(* Logix 5000 project; controller APM vendor 1 type 14 code 156 rev 30.11; software revision 30.00 *)

TASK MainTask (continuous, watchdog 500 ms) : MainProgram

MODULES
   Local : vendor 1 type 14 code 156 (Compact 0, rev 30.11)
END_MODULES

PROGRAM MainProgram   (* main routine MainRoutine *)
VAR
   CT_ACT_CT0 : BOOL;
   CT_ACT_CT1 : BOOL;
   CT_ACT_CT2 : BOOL;
   CT_ACT_CT3 : BOOL;
   CT_ACT_CT4 : BOOL;
   CT_ACT_CT5 : BOOL;
   CT_ACT_CT6 : BOOL;
   CT_ACT_HOM0 : BOOL;
   CT_ACT_HOM1 : BOOL;
   CT_ACT_HOM2 : BOOL;
   CT_ACT_HOM3 : BOOL;
   CT_ACT_STP : BOOL;
   CT_CA_AVC : BOOL;
   CT_CA_RET : BOOL;
   CT_CC_AVC : BOOL;
   CT_CC_RET : BOOL;
   CT_CNT1 : COUNTER := (PRE := 4);
   CT_CP_AVC : BOOL;
   CT_CP_RET : BOOL;
   CT_DIST : REAL;
   CT_ISOVER : BOOL;
   CT_MOT_M000 : BOOL;
   CT_MOT_M024 : BOOL;
   CT_MOT_M072 : BOOL;
   CT_MOT_M260 : BOOL;
   CT_OK : BOOL;
   CT_PBT_ESTP : BOOL;
   CT_PBT_HOM : BOOL;
   CT_PBT_STA : BOOL;
   CT_SEN_CaAvc : BOOL;
   CT_SEN_CaRet : BOOL;
   CT_SEN_CcAvc : BOOL;
   CT_SEN_CcRet : BOOL;
   CT_SEN_CpAvc : BOOL;
   CT_SEN_CpRet : BOOL;
   CT_SEN_D000 : BOOL;
   CT_SEN_D024 : BOOL;
   CT_SEN_D072 : BOOL;
   CT_SEN_D260 : BOOL;
   CT_SEN_MAT : BOOL;
   MAIN_ACTIVE : BOOL;
   MAIN_PBT_ESTP : BOOL;
   MAIN_PBT_STA : BOOL;
   PNT_ACT_0 : BOOL;
   PNT_ACT_1 : BOOL;
   PNT_ACT_2 : BOOL;
   PNT_ACT_3 : BOOL;
   PNT_ACT_4 : BOOL;
   PNT_ACT_HOM : BOOL;
   PNT_ACT_STP : BOOL;
   PNT_CNT1 : COUNTER := (PRE := 3);
   PNT_ISHOM : BOOL;
   PNT_ISOVER : BOOL;
   PNT_MTA_AVC : BOOL;
   PNT_MTA_RET : BOOL;
   PNT_MTB_AVC : BOOL;
   PNT_MTB_RET : BOOL;
   PNT_MTC_AVC : BOOL;
   PNT_MTC_RET : BOOL;
   PNT_PBT_HOM : BOOL;
   PNT_PBT_STA : BOOL;
   PNT_PBT_STP : BOOL;
   PNT_SEN_MAT : BOOL;
   PNT_SNA_AVC : BOOL;
   PNT_SNA_RET : BOOL;
   PNT_SNB_AVC : BOOL;
   PNT_SNB_RET : BOOL;
   PNT_SNC_AVC : BOOL;
   PNT_SNC_INT : BOOL;
   PNT_SNC_RET : BOOL;
END_VAR

ROUTINE Corte_actions   (* ladder *)
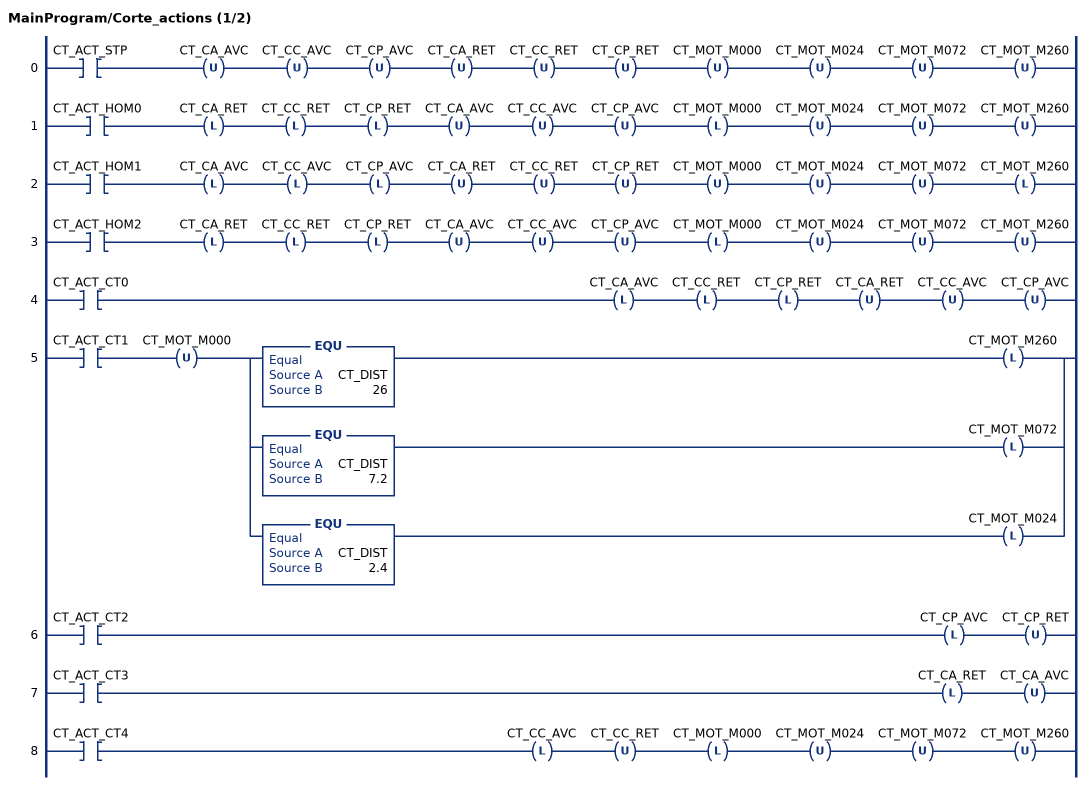
   0: XIC(CT_ACT_STP)OTU(CT_CA_AVC)OTU(CT_CC_AVC)OTU(CT_CP_AVC)OTU(CT_CA_RET)OTU(CT_CC_RET)OTU(CT_CP_RET)OTU(CT_MOT_M000)OTU(CT_MOT_M024)OTU(CT_MOT_M072)OTU(CT_MOT_M260);
   1: XIC(CT_ACT_HOM0)OTL(CT_CA_RET)OTL(CT_CC_RET)OTL(CT_CP_RET)OTU(CT_CA_AVC)OTU(CT_CC_AVC)OTU(CT_CP_AVC)OTL(CT_MOT_M000)OTU(CT_MOT_M024)OTU(CT_MOT_M072)OTU(CT_MOT_M260);
   2: XIC(CT_ACT_HOM1)OTL(CT_CA_AVC)OTL(CT_CC_AVC)OTL(CT_CP_AVC)OTU(CT_CA_RET)OTU(CT_CC_RET)OTU(CT_CP_RET)OTU(CT_MOT_M000)OTU(CT_MOT_M024)OTU(CT_MOT_M072)OTL(CT_MOT_M260);
   3: XIC(CT_ACT_HOM2)OTL(CT_CA_RET)OTL(CT_CC_RET)OTL(CT_CP_RET)OTU(CT_CA_AVC)OTU(CT_CC_AVC)OTU(CT_CP_AVC)OTL(CT_MOT_M000)OTU(CT_MOT_M024)OTU(CT_MOT_M072)OTU(CT_MOT_M260);
   4: XIC(CT_ACT_CT0)OTL(CT_CA_AVC)OTL(CT_CC_RET)OTL(CT_CP_RET)OTU(CT_CA_RET)OTU(CT_CC_AVC)OTU(CT_CP_AVC);
   5: XIC(CT_ACT_CT1)OTU(CT_MOT_M000)[EQU(CT_DIST,26) OTL(CT_MOT_M260) ,EQU(CT_DIST,7.2) OTL(CT_MOT_M072) ,EQU(CT_DIST,2.4) OTL(CT_MOT_M024) ];
   6: XIC(CT_ACT_CT2)OTL(CT_CP_AVC)OTU(CT_CP_RET);
   7: XIC(CT_ACT_CT3)OTL(CT_CA_RET)OTU(CT_CA_AVC);
   8: XIC(CT_ACT_CT4)OTL(CT_CC_AVC)OTU(CT_CC_RET)OTL(CT_MOT_M000)OTU(CT_MOT_M024)OTU(CT_MOT_M072)OTU(CT_MOT_M260);
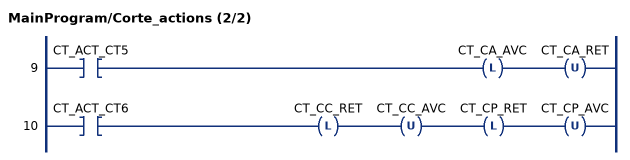
   9: XIC(CT_ACT_CT5)OTL(CT_CA_AVC)OTU(CT_CA_RET);
   10: XIC(CT_ACT_CT6)OTL(CT_CC_RET)OTU(CT_CC_AVC)OTL(CT_CP_RET)OTU(CT_CP_AVC);
END_ROUTINE

ROUTINE Corte_logic   (* ladder *)
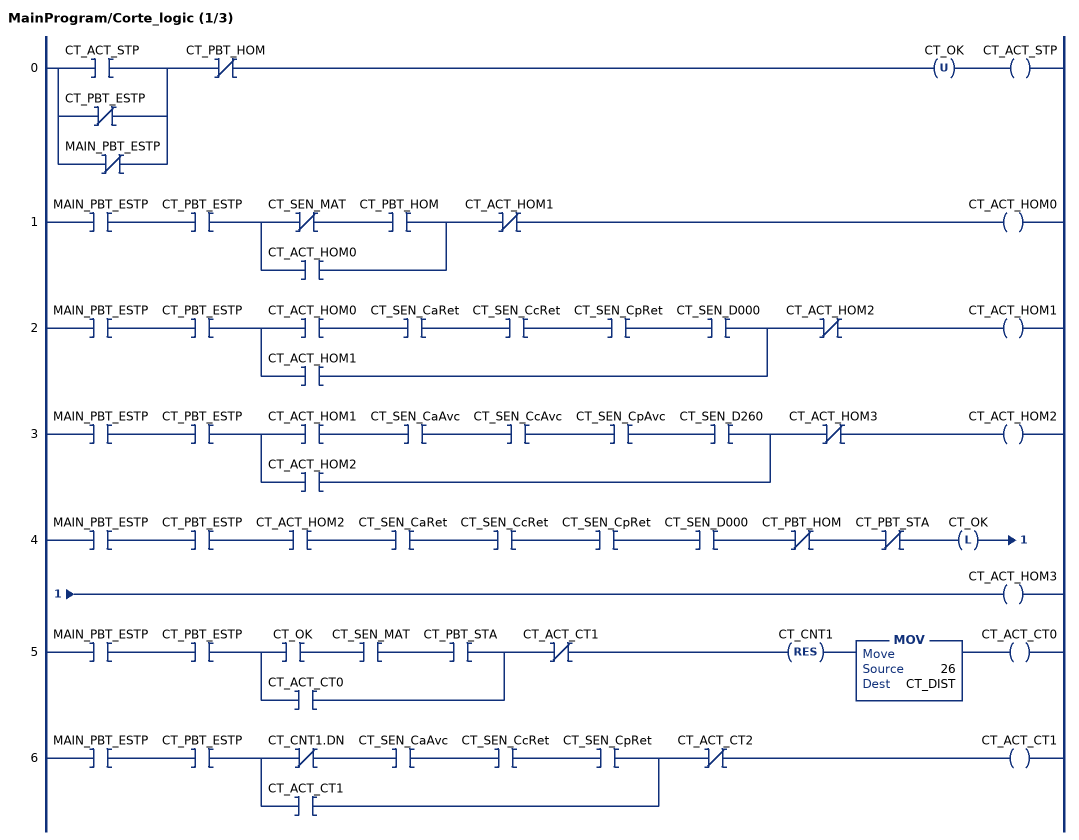
   0: [XIC(CT_ACT_STP) ,XIO(CT_PBT_ESTP) ,XIO(MAIN_PBT_ESTP) ]XIO(CT_PBT_HOM)OTU(CT_OK)OTE(CT_ACT_STP);
   1: XIC(MAIN_PBT_ESTP)XIC(CT_PBT_ESTP)[XIO(CT_SEN_MAT) XIC(CT_PBT_HOM) ,XIC(CT_ACT_HOM0) ]XIO(CT_ACT_HOM1)OTE(CT_ACT_HOM0);
   2: XIC(MAIN_PBT_ESTP)XIC(CT_PBT_ESTP)[XIC(CT_ACT_HOM0) XIC(CT_SEN_CaRet) XIC(CT_SEN_CcRet) XIC(CT_SEN_CpRet) XIC(CT_SEN_D000) ,XIC(CT_ACT_HOM1) ]XIO(CT_ACT_HOM2)OTE(CT_ACT_HOM1);
   3: XIC(MAIN_PBT_ESTP)XIC(CT_PBT_ESTP)[XIC(CT_ACT_HOM1) XIC(CT_SEN_CaAvc) XIC(CT_SEN_CcAvc) XIC(CT_SEN_CpAvc) XIC(CT_SEN_D260) ,XIC(CT_ACT_HOM2) ]XIO(CT_ACT_HOM3)OTE(CT_ACT_HOM2);
   4: XIC(MAIN_PBT_ESTP)XIC(CT_PBT_ESTP)XIC(CT_ACT_HOM2)XIC(CT_SEN_CaRet)XIC(CT_SEN_CcRet)XIC(CT_SEN_CpRet)XIC(CT_SEN_D000)XIO(CT_PBT_HOM)XIO(CT_PBT_STA)OTL(CT_OK)OTE(CT_ACT_HOM3);
   5: XIC(MAIN_PBT_ESTP)XIC(CT_PBT_ESTP)[XIC(CT_OK) XIC(CT_SEN_MAT) XIC(CT_PBT_STA) ,XIC(CT_ACT_CT0) ]XIO(CT_ACT_CT1)RES(CT_CNT1)MOV(26,CT_DIST)OTE(CT_ACT_CT0);
   6: XIC(MAIN_PBT_ESTP)XIC(CT_PBT_ESTP)[XIO(CT_CNT1.DN) XIC(CT_SEN_CaAvc) XIC(CT_SEN_CcRet) XIC(CT_SEN_CpRet) ,XIC(CT_ACT_CT1) ]XIO(CT_ACT_CT2)OTE(CT_ACT_CT1);
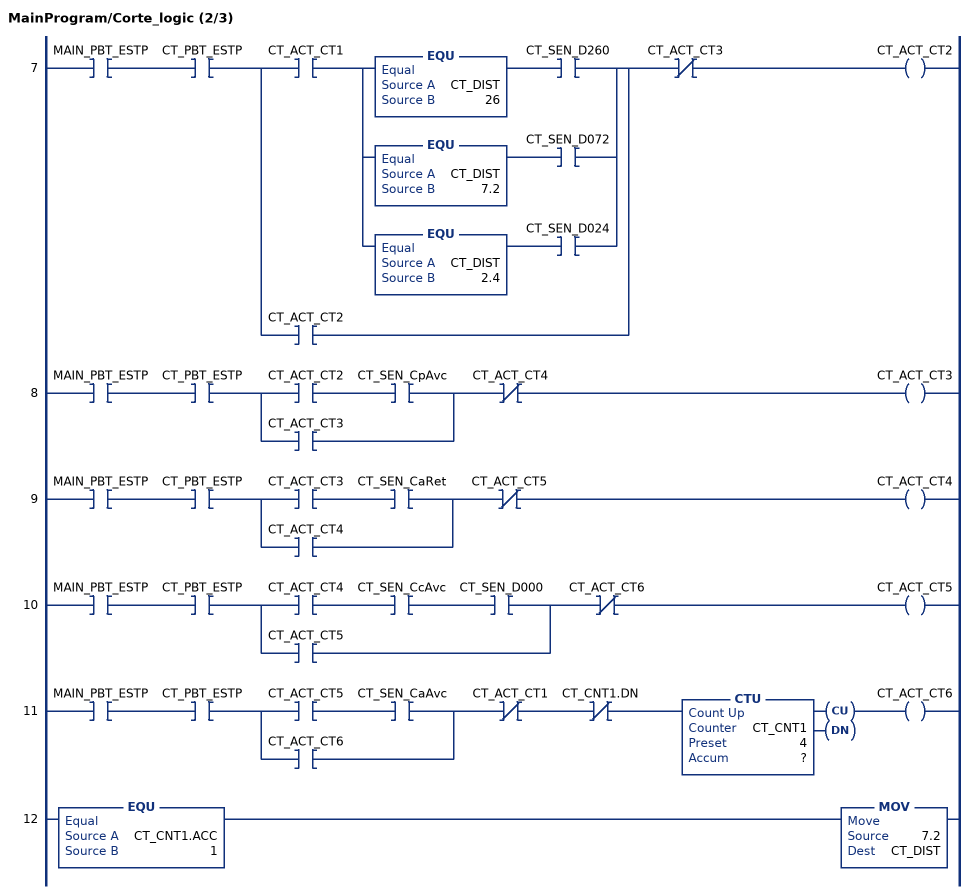
   7: XIC(MAIN_PBT_ESTP)XIC(CT_PBT_ESTP)[XIC(CT_ACT_CT1) [EQU(CT_DIST,26) XIC(CT_SEN_D260) ,EQU(CT_DIST,7.2) XIC(CT_SEN_D072) ,EQU(CT_DIST,2.4) XIC(CT_SEN_D024) ] ,XIC(CT_ACT_CT2) ]XIO(CT_ACT_CT3)OTE(CT_ACT_CT2);
   8: XIC(MAIN_PBT_ESTP)XIC(CT_PBT_ESTP)[XIC(CT_ACT_CT2) XIC(CT_SEN_CpAvc) ,XIC(CT_ACT_CT3) ]XIO(CT_ACT_CT4)OTE(CT_ACT_CT3);
   9: XIC(MAIN_PBT_ESTP)XIC(CT_PBT_ESTP)[XIC(CT_ACT_CT3) XIC(CT_SEN_CaRet) ,XIC(CT_ACT_CT4) ]XIO(CT_ACT_CT5)OTE(CT_ACT_CT4);
   10: XIC(MAIN_PBT_ESTP)XIC(CT_PBT_ESTP)[XIC(CT_ACT_CT4) XIC(CT_SEN_CcAvc) XIC(CT_SEN_D000) ,XIC(CT_ACT_CT5) ]XIO(CT_ACT_CT6)OTE(CT_ACT_CT5);
   11: XIC(MAIN_PBT_ESTP)XIC(CT_PBT_ESTP)[XIC(CT_ACT_CT5) XIC(CT_SEN_CaAvc) ,XIC(CT_ACT_CT6) ]XIO(CT_ACT_CT1)XIO(CT_CNT1.DN)CTU(CT_CNT1,?,?)OTE(CT_ACT_CT6);
   12: EQU(CT_CNT1.ACC,1)MOV(7.2,CT_DIST);
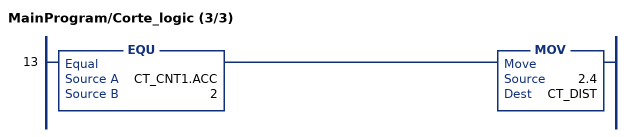
   13: EQU(CT_CNT1.ACC,2)MOV(2.4,CT_DIST);
END_ROUTINE

ROUTINE MainRoutine   (* ladder *)
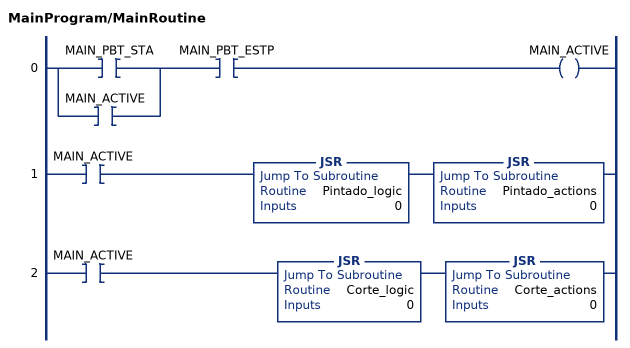
   0: [XIC(MAIN_PBT_STA) ,XIC(MAIN_ACTIVE) ]XIC(MAIN_PBT_ESTP)OTE(MAIN_ACTIVE);
   1: XIC(MAIN_ACTIVE)JSR(Pintado_logic,0)JSR(Pintado_actions,0);
   2: XIC(MAIN_ACTIVE)JSR(Corte_logic,0)JSR(Corte_actions,0);
END_ROUTINE

ROUTINE Pintado_actions   (* ladder *)
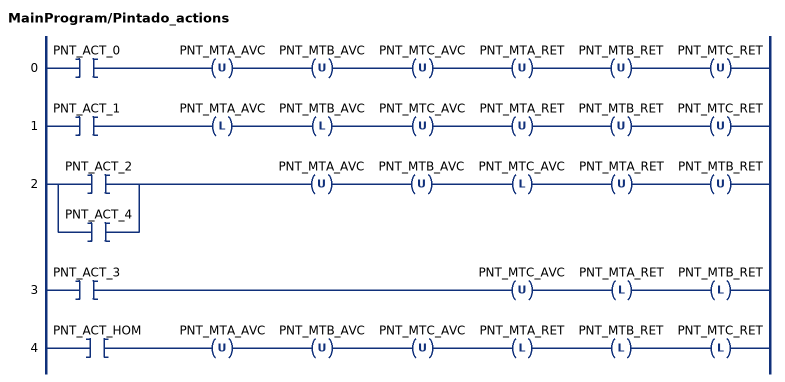
   0: XIC(PNT_ACT_0)OTU(PNT_MTA_AVC)OTU(PNT_MTB_AVC)OTU(PNT_MTC_AVC)OTU(PNT_MTA_RET)OTU(PNT_MTB_RET)OTU(PNT_MTC_RET);
   1: XIC(PNT_ACT_1)OTL(PNT_MTA_AVC)OTL(PNT_MTB_AVC)OTU(PNT_MTC_AVC)OTU(PNT_MTA_RET)OTU(PNT_MTB_RET)OTU(PNT_MTC_RET);
   2: [XIC(PNT_ACT_2) ,XIC(PNT_ACT_4) ]OTU(PNT_MTA_AVC)OTU(PNT_MTB_AVC)OTL(PNT_MTC_AVC)OTU(PNT_MTA_RET)OTU(PNT_MTB_RET);
   3: XIC(PNT_ACT_3)OTU(PNT_MTC_AVC)OTL(PNT_MTA_RET)OTL(PNT_MTB_RET);
   4: XIC(PNT_ACT_HOM)OTU(PNT_MTA_AVC)OTU(PNT_MTB_AVC)OTU(PNT_MTC_AVC)OTL(PNT_MTA_RET)OTL(PNT_MTB_RET)OTL(PNT_MTC_RET);
END_ROUTINE

ROUTINE Pintado_logic   (* ladder *)
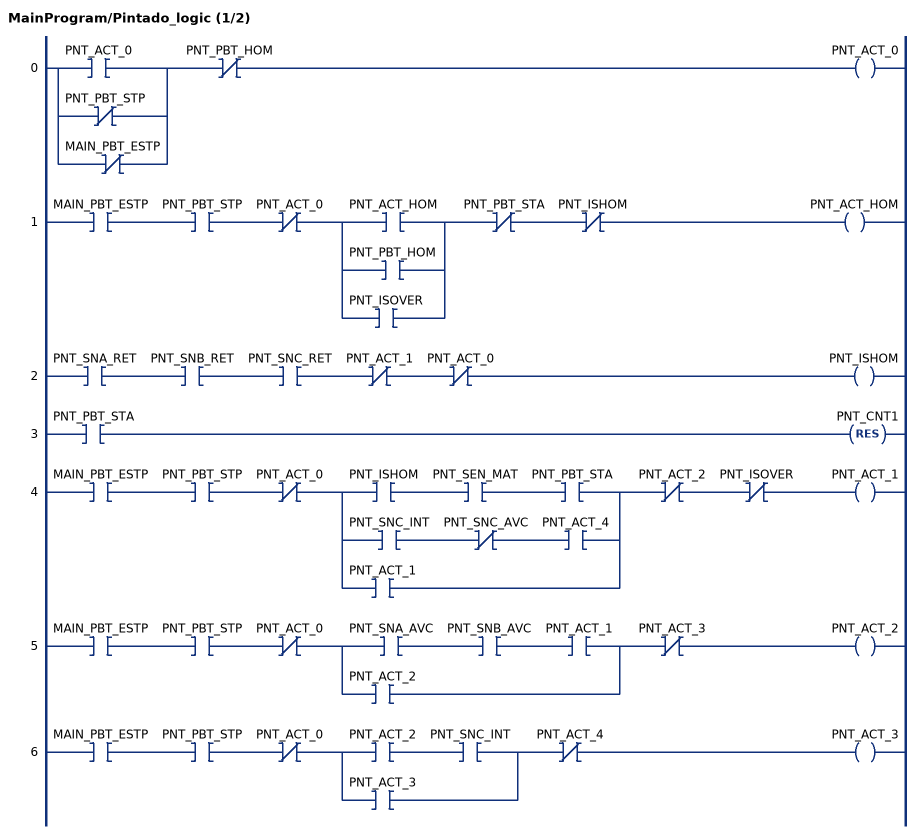
   0: [XIC(PNT_ACT_0) ,XIO(PNT_PBT_STP) ,XIO(MAIN_PBT_ESTP) ]XIO(PNT_PBT_HOM)OTE(PNT_ACT_0);
   1: XIC(MAIN_PBT_ESTP)XIC(PNT_PBT_STP)XIO(PNT_ACT_0)[XIC(PNT_ACT_HOM) ,XIC(PNT_PBT_HOM) ,XIC(PNT_ISOVER) ]XIO(PNT_PBT_STA)XIO(PNT_ISHOM)OTE(PNT_ACT_HOM);
   2: XIC(PNT_SNA_RET)XIC(PNT_SNB_RET)XIC(PNT_SNC_RET)XIO(PNT_ACT_1)XIO(PNT_ACT_0)OTE(PNT_ISHOM);
   3: XIC(PNT_PBT_STA)RES(PNT_CNT1);
   4: XIC(MAIN_PBT_ESTP)XIC(PNT_PBT_STP)XIO(PNT_ACT_0)[XIC(PNT_ISHOM) XIC(PNT_SEN_MAT) XIC(PNT_PBT_STA) ,XIC(PNT_SNC_INT) XIO(PNT_SNC_AVC) XIC(PNT_ACT_4) ,XIC(PNT_ACT_1) ]XIO(PNT_ACT_2)XIO(PNT_ISOVER)OTE(PNT_ACT_1);
   5: XIC(MAIN_PBT_ESTP)XIC(PNT_PBT_STP)XIO(PNT_ACT_0)[XIC(PNT_SNA_AVC) XIC(PNT_SNB_AVC) XIC(PNT_ACT_1) ,XIC(PNT_ACT_2) ]XIO(PNT_ACT_3)OTE(PNT_ACT_2);
   6: XIC(MAIN_PBT_ESTP)XIC(PNT_PBT_STP)XIO(PNT_ACT_0)[XIC(PNT_ACT_2) XIC(PNT_SNC_INT) ,XIC(PNT_ACT_3) ]XIO(PNT_ACT_4)OTE(PNT_ACT_3);
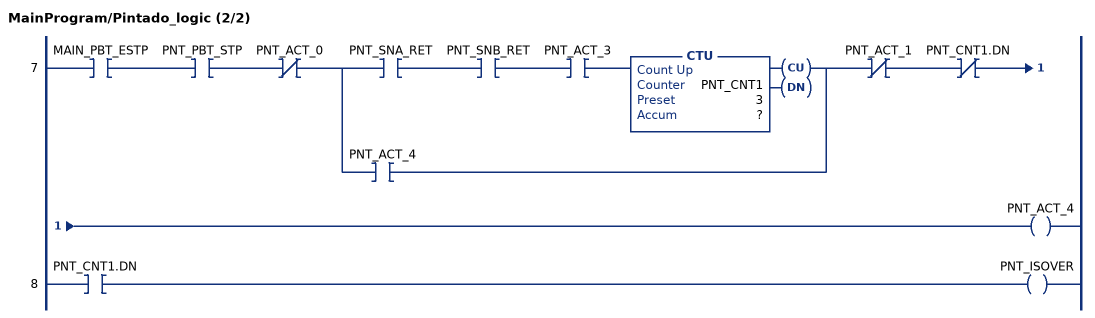
   7: XIC(MAIN_PBT_ESTP)XIC(PNT_PBT_STP)XIO(PNT_ACT_0)[XIC(PNT_SNA_RET) XIC(PNT_SNB_RET) XIC(PNT_ACT_3) CTU(PNT_CNT1,?,?) ,XIC(PNT_ACT_4) ]XIO(PNT_ACT_1)XIO(PNT_CNT1.DN)OTE(PNT_ACT_4);
   8: XIC(PNT_CNT1.DN)OTE(PNT_ISOVER);
END_ROUTINE
END_PROGRAM
